(* Logix 5000 project; controller Carpenter_Meter_SCP vendor 1 type 14 code 217 rev 31.11; software revision 31.01; part 2 of 7 *)

ADD_ON_INSTRUCTION TGE_AI   (* revision 0.0, vendor Tallgrass Energy *)
VAR_IN_OUT
   UDT : TGE_AI_UDT; {required}
END_VAR
VAR_INPUT
   Raw : REAL; {required}   // Raw Data
END_VAR
VAR_OUTPUT
   EU : REAL; {access Read Only, visible}   // Scaled Value in Engineering Units
   Avg : REAL; {access Read Only, visible}   // Average value
   MalfAlm : BOOL; {access Read Only, visible}   // Signal Malfunction Alarm Status
   HAlm : BOOL; {access Read Only, visible}   // High Alarm status
   HHAlm : BOOL; {access Read Only, visible}   // High High Alarm status
   LAlm : BOOL; {access Read Only, visible}   // Low Alarm status
   LLAlm : BOOL; {access Read Only, visible}   // Low low Alarm status
   ROCNegAlm : BOOL; {access Read Only, visible}   // Negative Rate Of Change Alarm status
   ROCPosAlm : BOOL; {access Read Only, visible}   // Positive Rate Of Change Alarm status
   Percent : REAL; {access Read Only, visible}   // Percent of Engineering
END_VAR
VAR
   HHActive : BOOL;   // High High Alarm Active
   HActive : BOOL;   // High Alarm Active
   LActive : BOOL;   // Low Alarm Active
   LLActive : BOOL;   // Low Low Alarm Active
   RocAlm : TGE_ROC;
   MaxPriority : DINT; {access None}
END_VAR

ROUTINE Logic   (* ladder *)
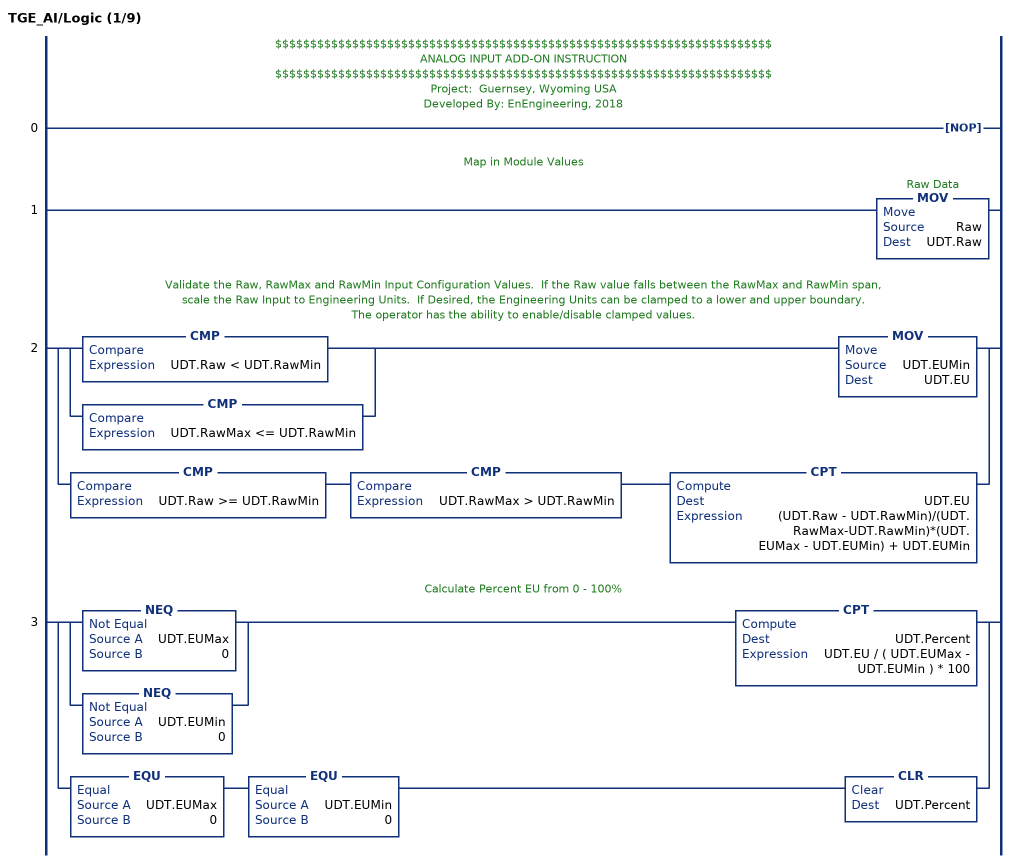
   // $$$$$$$$$$$$$$$$$$$$$$$$$$$$$$$$$$$$$$$$$$$$$$$$$$$$$$$$$$$$$$$$$$$$$$$
   // ANALOG INPUT ADD-ON INSTRUCTION
   // $$$$$$$$$$$$$$$$$$$$$$$$$$$$$$$$$$$$$$$$$$$$$$$$$$$$$$$$$$$$$$$$$$$$$$$
   // Project:  Guernsey, Wyoming USA
   // Developed By: EnEngineering, 2018
   0: NOP();
   // Map in Module Values
   1: MOV(Raw,UDT.Raw);
   // Validate the Raw, RawMax and RawMin Input Configuration Values.  If the Raw value falls between the RawMax and RawMin span,
   // scale the Raw Input to Engineering Units.  If Desired, the Engineering Units can be clamped to a lower and upper boundary.
   // The operator has the ability to enable/disable clamped values.
   2: [[CMP(UDT.Raw < UDT.RawMin) ,CMP(UDT.RawMax <= UDT.RawMin) ] MOV(UDT.EUMin,UDT.EU) ,CMP(UDT.Raw >= UDT.RawMin) CMP(UDT.RawMax > UDT.RawMin) CPT(UDT.EU,(UDT.Raw - UDT.RawMin)/(UDT.RawMax-UDT.RawMin)*(UDT.EUMax - UDT.EUMin) + UDT.EUMin) ];
   // Calculate Percent EU from 0 - 100%
   3: [[NEQ(UDT.EUMax,0) ,NEQ(UDT.EUMin,0) ] CPT(UDT.Percent,UDT.EU / ( UDT.EUMax - UDT.EUMin ) * 100) ,EQU(UDT.EUMax,0) EQU(UDT.EUMin,0) CLR(UDT.Percent) ];
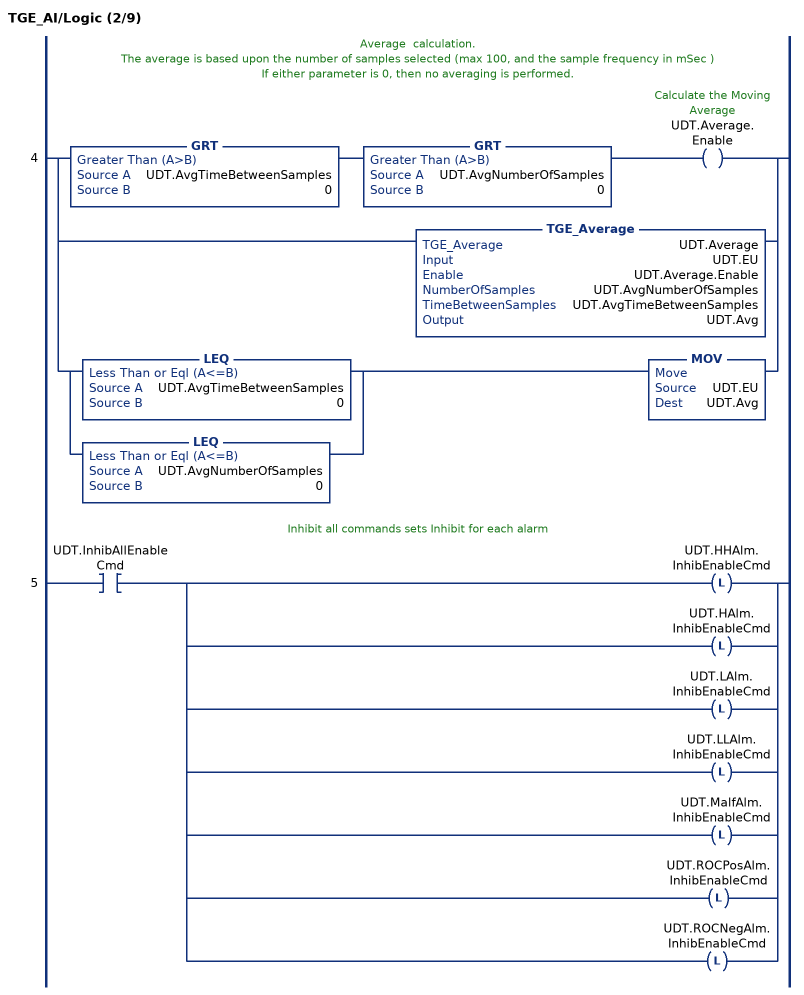
   // Average  calculation.
   // The average is based upon the number of samples selected (max 100, and the sample frequency in mSec )
   // If either parameter is 0, then no averaging is performed.
   4: [GRT(UDT.AvgTimeBetweenSamples,0) GRT(UDT.AvgNumberOfSamples,0) OTE(UDT.Average.Enable) ,TGE_Average(UDT.Average,UDT.EU,UDT.Average.Enable,UDT.AvgNumberOfSamples,UDT.AvgTimeBetweenSamples,UDT.Avg) ,[LEQ(UDT.AvgTimeBetweenSamples,0) ,LEQ(UDT.AvgNumberOfSamples,0) ] MOV(UDT.EU,UDT.Avg) ];
   // Inhibit all commands sets Inhibit for each alarm
   5: XIC(UDT.InhibAllEnableCmd)[OTL(UDT.HHAlm.InhibEnableCmd) ,OTL(UDT.HAlm.InhibEnableCmd) ,OTL(UDT.LAlm.InhibEnableCmd) ,OTL(UDT.LLAlm.InhibEnableCmd) ,OTL(UDT.MalfAlm.InhibEnableCmd) ,OTL(UDT.ROCPosAlm.InhibEnableCmd) ,OTL(UDT.ROCNegAlm.InhibEnableCmd) ];
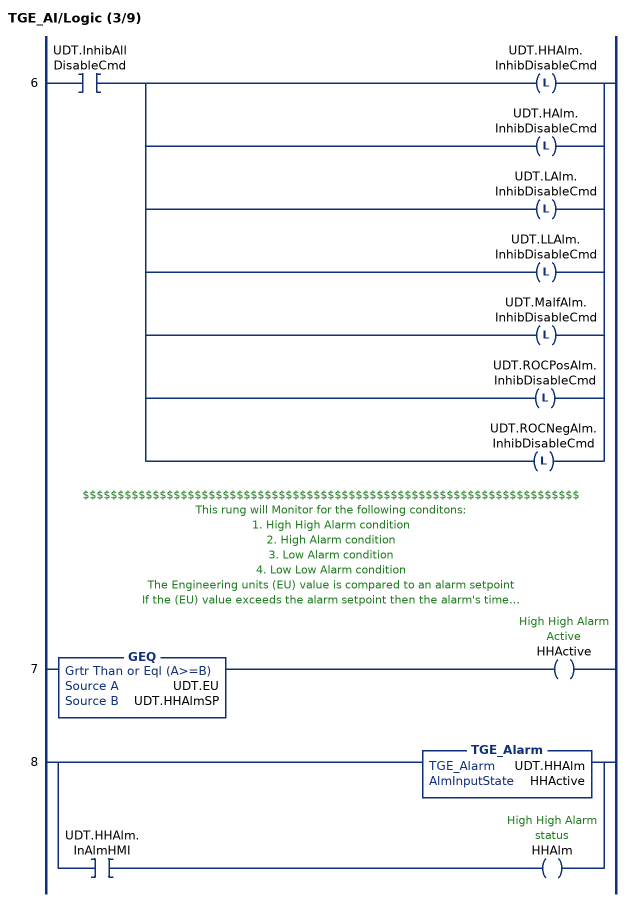
   6: XIC(UDT.InhibAllDisableCmd)[OTL(UDT.HHAlm.InhibDisableCmd) ,OTL(UDT.HAlm.InhibDisableCmd) ,OTL(UDT.LAlm.InhibDisableCmd) ,OTL(UDT.LLAlm.InhibDisableCmd) ,OTL(UDT.MalfAlm.InhibDisableCmd) ,OTL(UDT.ROCPosAlm.InhibDisableCmd) ,OTL(UDT.ROCNegAlm.InhibDisableCmd) ];
   // $$$$$$$$$$$$$$$$$$$$$$$$$$$$$$$$$$$$$$$$$$$$$$$$$$$$$$$$$$$$$$$$$$$$$$$
   //  This rung will Monitor for the following conditons:
   // 1. High High Alarm condition
   // 2. High Alarm condition
   // 3. Low Alarm condition
   // 4. Low Low Alarm condition
   // The Engineering units (EU) value is compared to an alarm setpoint
   //  If the (EU) value exceeds the alarm setpoint then the alarm's timer
   // preset value is loaded and the Alarm's Active bit is set
   // Note: The Preset value of this timer is configured via the udt
   // The alarm's Active bit is used as the Input to the aoiAlarm instruction.
   // The aoiAlarm's Alm bit is then used to update the Alarm status bit
   // $$$$$$$$$$$$$$$$$$$$$$$$$$$$$$$$$$$$$$$$$$$$$$$$$$$$$$$$$$$$$$$$$$$$$$$
   7: GEQ(UDT.EU,UDT.HHAlmSP)OTE(HHActive);
   8: [TGE_Alarm(UDT.HHAlm,HHActive) ,XIC(UDT.HHAlm.InAlmHMI) OTE(HHAlm) ];
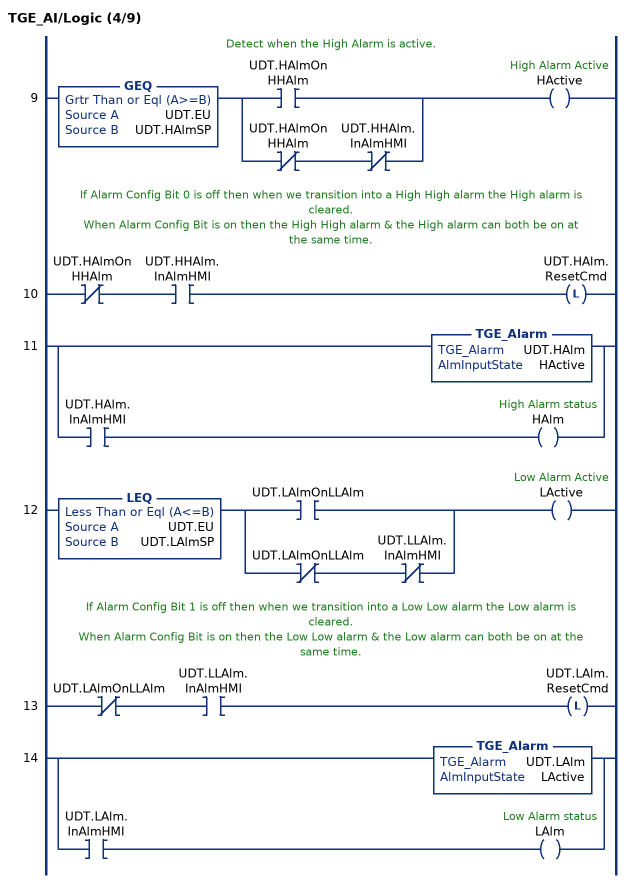
   // Detect when the High Alarm is active.
   9: GEQ(UDT.EU,UDT.HAlmSP)[XIC(UDT.HAlmOnHHAlm) ,XIO(UDT.HAlmOnHHAlm) XIO(UDT.HHAlm.InAlmHMI) ]OTE(HActive);
   // If Alarm Config Bit 0 is off then when we transition into a High High alarm the High alarm is cleared.
   // When Alarm Config Bit is on then the High High alarm & the High alarm can both be on at the same time.
   10: XIO(UDT.HAlmOnHHAlm)XIC(UDT.HHAlm.InAlmHMI)OTL(UDT.HAlm.ResetCmd);
   11: [TGE_Alarm(UDT.HAlm,HActive) ,XIC(UDT.HAlm.InAlmHMI) OTE(HAlm) ];
   12: LEQ(UDT.EU,UDT.LAlmSP)[XIC(UDT.LAlmOnLLAlm) ,XIO(UDT.LAlmOnLLAlm) XIO(UDT.LLAlm.InAlmHMI) ]OTE(LActive);
   // If Alarm Config Bit 1 is off then when we transition into a Low Low alarm the Low alarm is cleared.
   // When Alarm Config Bit is on then the Low Low alarm & the Low alarm can both be on at the same time.
   13: XIO(UDT.LAlmOnLLAlm)XIC(UDT.LLAlm.InAlmHMI)OTL(UDT.LAlm.ResetCmd);
   14: [TGE_Alarm(UDT.LAlm,LActive) ,XIC(UDT.LAlm.InAlmHMI) OTE(LAlm) ];
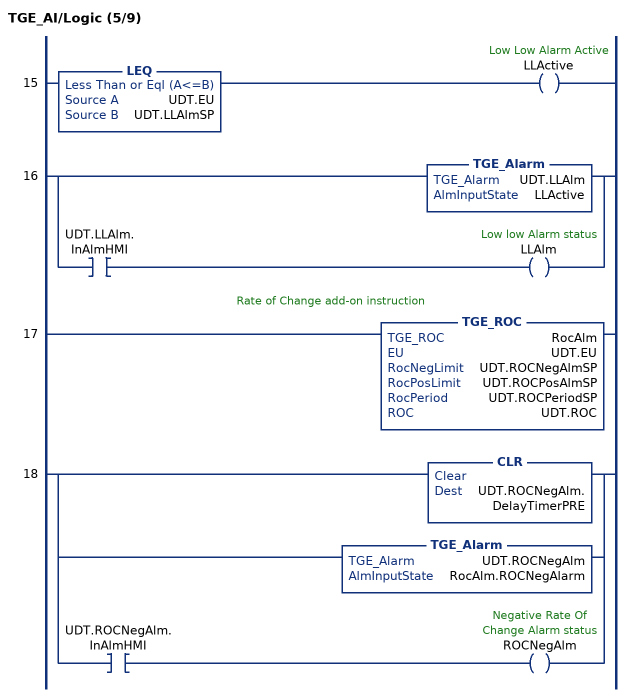
   15: LEQ(UDT.EU,UDT.LLAlmSP)OTE(LLActive);
   16: [TGE_Alarm(UDT.LLAlm,LLActive) ,XIC(UDT.LLAlm.InAlmHMI) OTE(LLAlm) ];
   // Rate of Change add-on instruction
   17: TGE_ROC(RocAlm,UDT.EU,UDT.ROCNegAlmSP,UDT.ROCPosAlmSP,UDT.ROCPeriodSP,UDT.ROC);
   18: [CLR(UDT.ROCNegAlm.DelayTimerPRE) ,TGE_Alarm(UDT.ROCNegAlm,RocAlm.ROCNegAlarm) ,XIC(UDT.ROCNegAlm.InAlmHMI) OTE(ROCNegAlm) ];
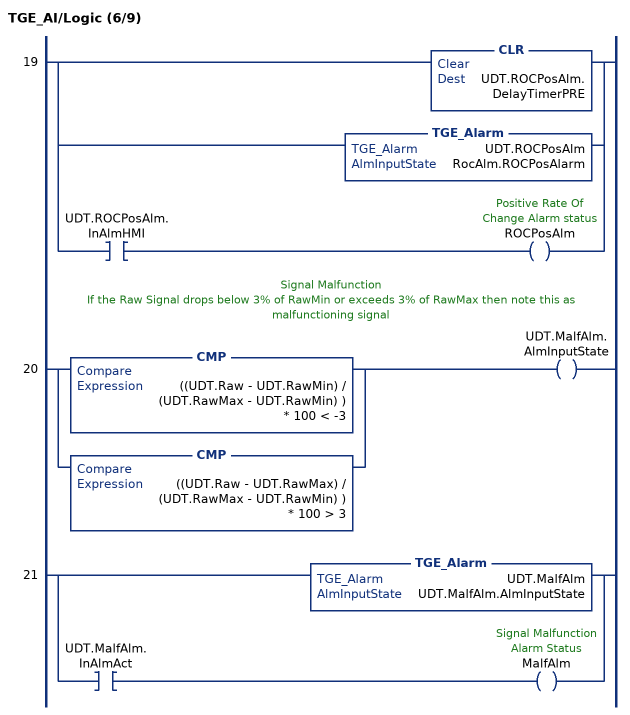
   19: [CLR(UDT.ROCPosAlm.DelayTimerPRE) ,TGE_Alarm(UDT.ROCPosAlm,RocAlm.ROCPosAlarm) ,XIC(UDT.ROCPosAlm.InAlmHMI) OTE(ROCPosAlm) ];
   // Signal Malfunction
   // If the Raw Signal drops below 3% of RawMin or exceeds 3% of RawMax then note this as malfunctioning signal
   20: [CMP(((UDT.Raw - UDT.RawMin) / (UDT.RawMax - UDT.RawMin) ) * 100 < -3) ,CMP(((UDT.Raw - UDT.RawMax) / (UDT.RawMax - UDT.RawMin) ) * 100 > 3) ]OTE(UDT.MalfAlm.AlmInputState);
   21: [TGE_Alarm(UDT.MalfAlm,UDT.MalfAlm.AlmInputState) ,XIC(UDT.MalfAlm.InAlmAct) OTE(MalfAlm) ];
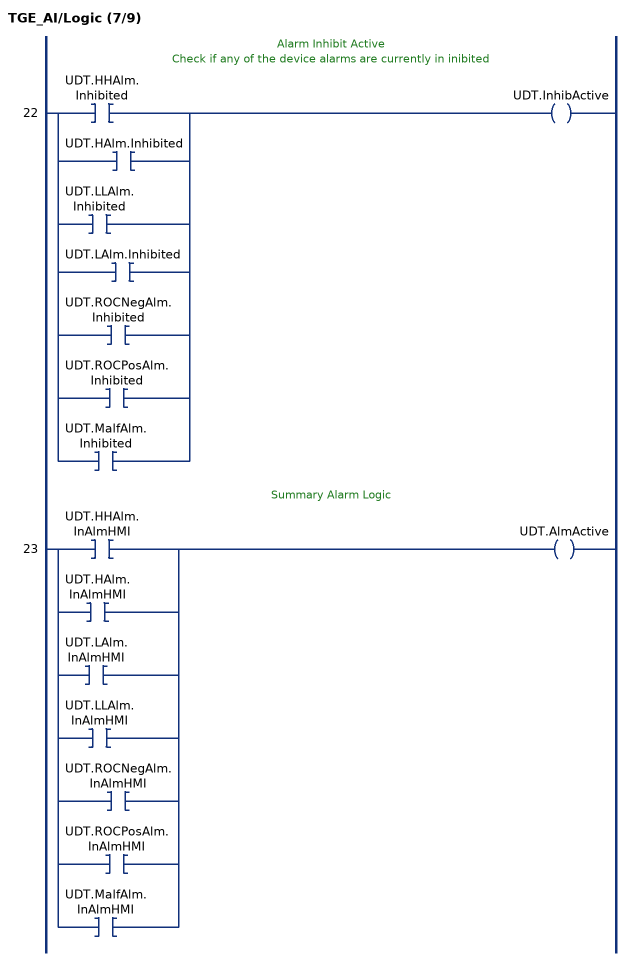
   // Alarm Inhibit Active
   // Check if any of the device alarms are currently in inibited
   22: [XIC(UDT.HHAlm.Inhibited) ,XIC(UDT.HAlm.Inhibited) ,XIC(UDT.LLAlm.Inhibited) ,XIC(UDT.LAlm.Inhibited) ,XIC(UDT.ROCNegAlm.Inhibited) ,XIC(UDT.ROCPosAlm.Inhibited) ,XIC(UDT.MalfAlm.Inhibited) ]OTE(UDT.InhibActive);
   // Summary Alarm Logic
   23: [XIC(UDT.HHAlm.InAlmHMI) ,XIC(UDT.HAlm.InAlmHMI) ,XIC(UDT.LAlm.InAlmHMI) ,XIC(UDT.LLAlm.InAlmHMI) ,XIC(UDT.ROCNegAlm.InAlmHMI) ,XIC(UDT.ROCPosAlm.InAlmHMI) ,XIC(UDT.MalfAlm.InAlmHMI) ]OTE(UDT.AlmActive);
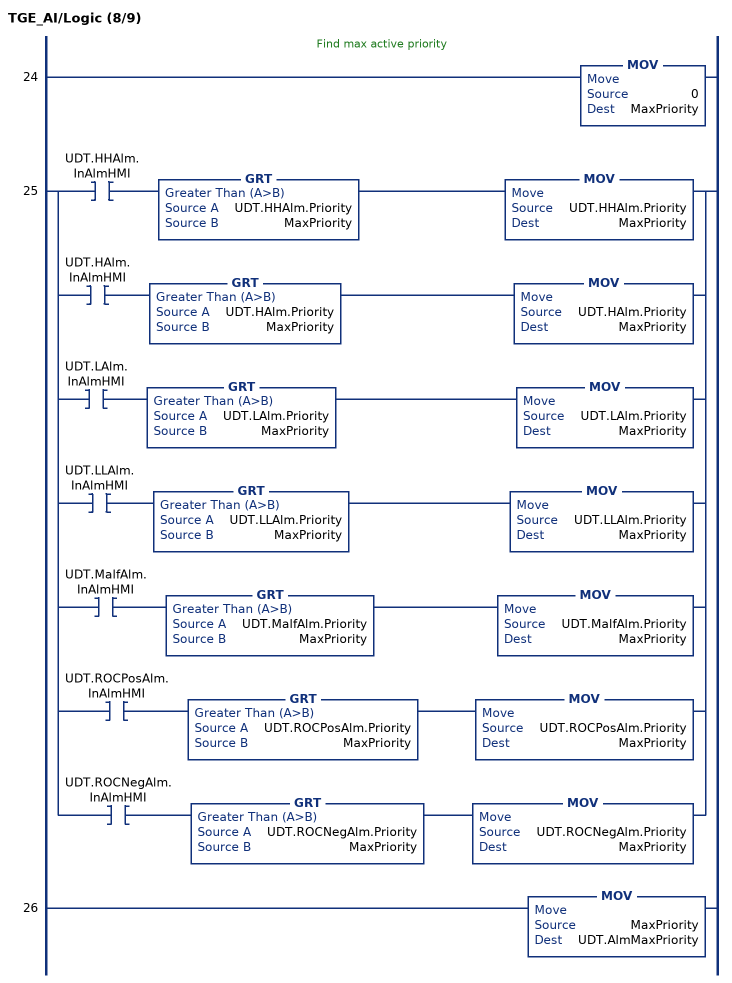
   // Find max active priority
   24: MOV(0,MaxPriority);
   25: [XIC(UDT.HHAlm.InAlmHMI) GRT(UDT.HHAlm.Priority,MaxPriority) MOV(UDT.HHAlm.Priority,MaxPriority) ,XIC(UDT.HAlm.InAlmHMI) GRT(UDT.HAlm.Priority,MaxPriority) MOV(UDT.HAlm.Priority,MaxPriority) ,XIC(UDT.LAlm.InAlmHMI) GRT(UDT.LAlm.Priority,MaxPriority) MOV(UDT.LAlm.Priority,MaxPriority) ,XIC(UDT.LLAlm.InAlmHMI) GRT(UDT.LLAlm.Priority,MaxPriority) MOV(UDT.LLAlm.Priority,MaxPriority) ,XIC(UDT.MalfAlm.InAlmHMI) GRT(UDT.MalfAlm.Priority,MaxPriority) MOV(UDT.MalfAlm.Priority,MaxPriority) ,XIC(UDT.ROCPosAlm.InAlmHMI) GRT(UDT.ROCPosAlm.Priority,MaxPriority) MOV(UDT.ROCPosAlm.Priority,MaxPriority) ,XIC(UDT.ROCNegAlm.InAlmHMI) GRT(UDT.ROCNegAlm.Priority,MaxPriority) MOV(UDT.ROCNegAlm.Priority,MaxPriority) ];
   26: MOV(MaxPriority,UDT.AlmMaxPriority);
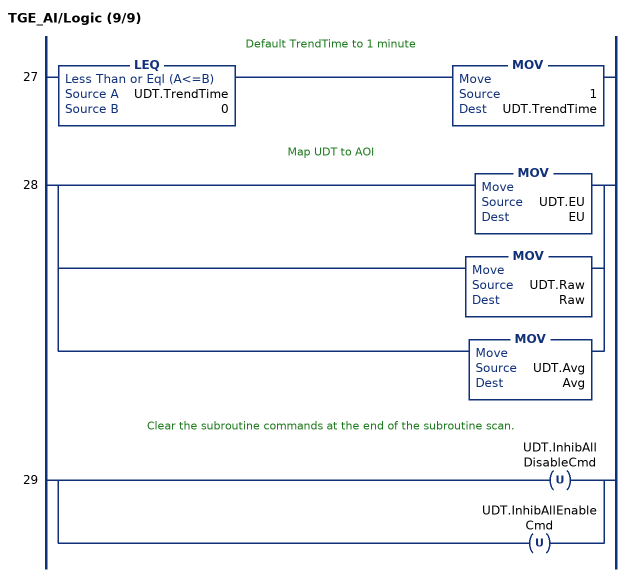
   // Default TrendTime to 1 minute
   27: LEQ(UDT.TrendTime,0)MOV(1,UDT.TrendTime);
   // Map UDT to AOI
   28: [MOV(UDT.EU,EU) ,MOV(UDT.Raw,Raw) ,MOV(UDT.Avg,Avg) ];
   // Clear the subroutine commands at the end of the subroutine scan.
   29: [OTU(UDT.InhibAllDisableCmd) ,OTU(UDT.InhibAllEnableCmd) ];
END_ROUTINE
END_ADD_ON_INSTRUCTION

ADD_ON_INSTRUCTION TGE_Alarm   (* revision 0.0, vendor Tallgrass Energy *)
VAR_INPUT
   EnableCmd : BOOL;
   DisableCmd : BOOL;
   ResetCmd : BOOL;
   TimerReset : BOOL;
   Enabled : BOOL; {visible}
   AckReq : BOOL;
   ResetReq : BOOL;
   AlmInputState : BOOL; {required}
   AckCmd : BOOL;
   AlmExists : BOOL := 1;
END_VAR
VAR_OUTPUT
   InAlmAct : BOOL; {visible}
END_VAR
VAR_INPUT
   InAlmHMI : BOOL;
END_VAR
VAR_OUTPUT
   Acked : BOOL;
END_VAR
VAR_INPUT
   DelayTimerPRE : REAL; {visible}
   ReminderTimerPRE : REAL; {visible}
END_VAR
VAR_OUTPUT
   ReminderFlag : BOOL; {visible}
   DelayTimerACC : REAL; {visible}
   ReminderTimerACC : REAL; {visible}
END_VAR
VAR_INPUT
   InhibEnableCmd : BOOL;
   InhibDisableCmd : BOOL;
END_VAR
VAR_OUTPUT
   Inhibited : BOOL;
   Priority : DINT; {visible}
END_VAR
VAR
   DelayTimer : TIMER;
   ReminderTimer : TIMER;
END_VAR

ROUTINE Logic   (* ladder *)
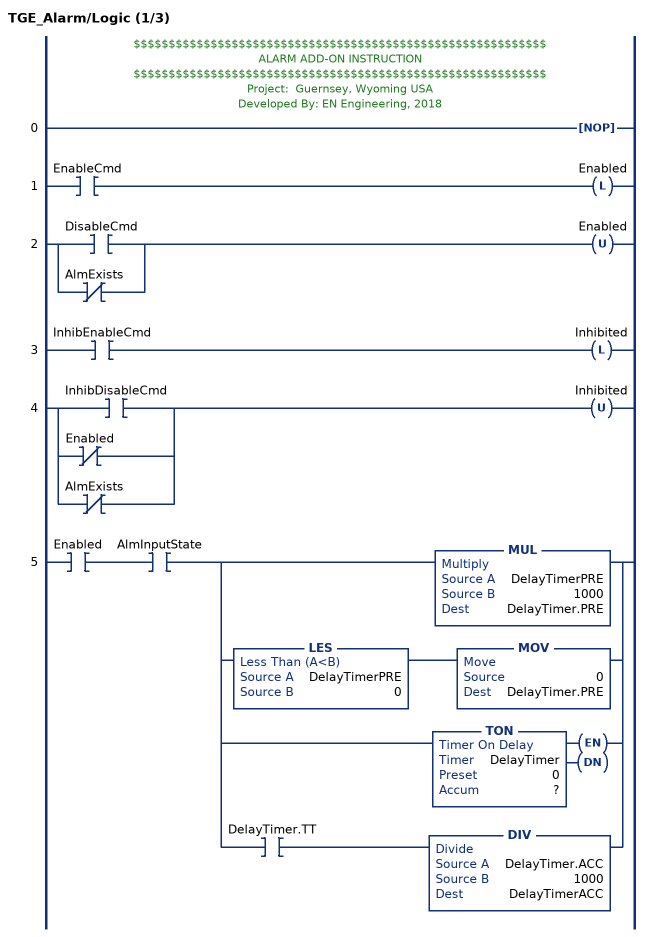
   // $$$$$$$$$$$$$$$$$$$$$$$$$$$$$$$$$$$$$$$$$$$$$$$$$$$$$$$$$$$
   // ALARM ADD-ON INSTRUCTION
   // $$$$$$$$$$$$$$$$$$$$$$$$$$$$$$$$$$$$$$$$$$$$$$$$$$$$$$$$$$$
   // Project:  Guernsey, Wyoming USA
   // Developed By: EN Engineering, 2018
   0: NOP();
   1: XIC(EnableCmd)OTL(Enabled);
   2: [XIC(DisableCmd) ,XIO(AlmExists) ]OTU(Enabled);
   3: XIC(InhibEnableCmd)OTL(Inhibited);
   4: [XIC(InhibDisableCmd) ,XIO(Enabled) ,XIO(AlmExists) ]OTU(Inhibited);
   5: XIC(Enabled)XIC(AlmInputState)[MUL(DelayTimerPRE,1000,DelayTimer.PRE) ,[LES(DelayTimerPRE,0) MOV(0,DelayTimer.PRE) ,TON(DelayTimer,?,?) ] ,XIC(DelayTimer.TT) DIV(DelayTimer.ACC,1000,DelayTimerACC) ];
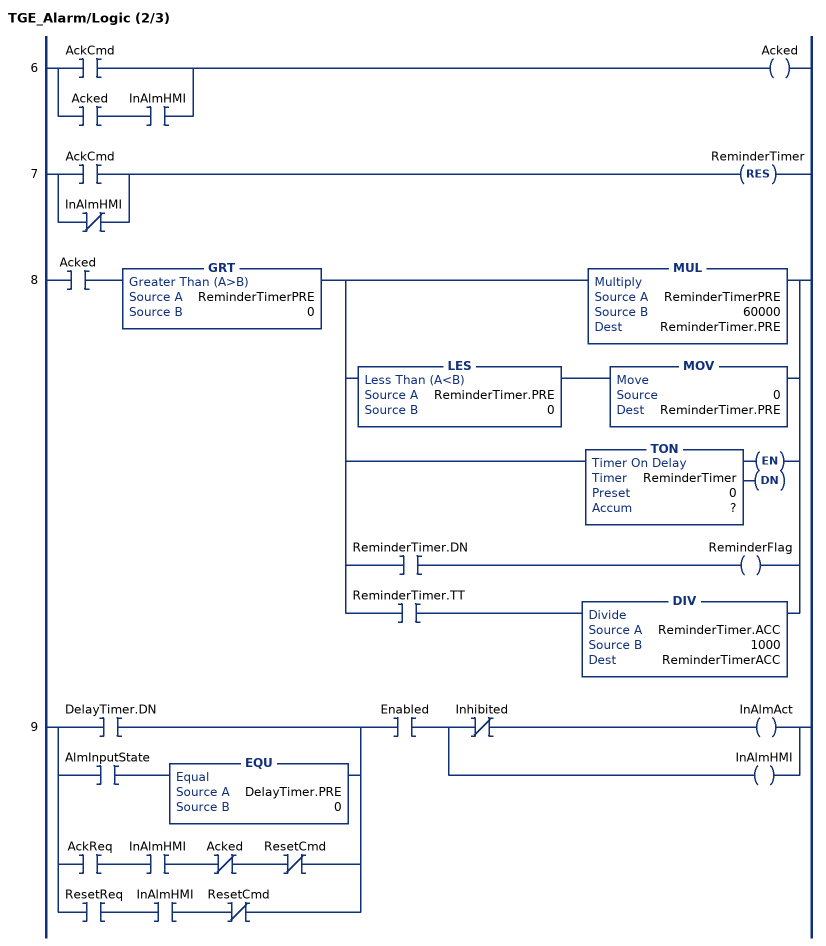
   6: [XIC(AckCmd) ,XIC(Acked) XIC(InAlmHMI) ]OTE(Acked);
   7: [XIC(AckCmd) ,XIO(InAlmHMI) ]RES(ReminderTimer);
   8: XIC(Acked)GRT(ReminderTimerPRE,0)[MUL(ReminderTimerPRE,60000,ReminderTimer.PRE) ,[LES(ReminderTimer.PRE,0) MOV(0,ReminderTimer.PRE) ,TON(ReminderTimer,?,?) ] ,XIC(ReminderTimer.DN) OTE(ReminderFlag) ,XIC(ReminderTimer.TT) DIV(ReminderTimer.ACC,1000,ReminderTimerACC) ];
   9: [[XIC(DelayTimer.DN) ,XIC(AlmInputState) EQU(DelayTimer.PRE,0) ] ,XIC(AckReq) XIC(InAlmHMI) XIO(Acked) XIO(ResetCmd) ,XIC(ResetReq) XIC(InAlmHMI) XIO(ResetCmd) ]XIC(Enabled)[XIO(Inhibited) OTE(InAlmAct) ,OTE(InAlmHMI) ];
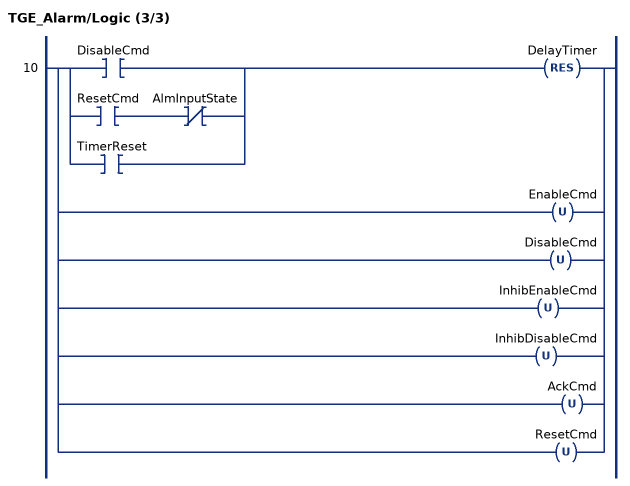
   10: [[XIC(DisableCmd) ,XIC(ResetCmd) XIO(AlmInputState) ,XIC(TimerReset) ] RES(DelayTimer) ,OTU(EnableCmd) ,OTU(DisableCmd) ,OTU(InhibEnableCmd) ,OTU(InhibDisableCmd) ,OTU(AckCmd) ,OTU(ResetCmd) ];
END_ROUTINE
END_ADD_ON_INSTRUCTION

ADD_ON_INSTRUCTION TGE_Average   (* revision 0.0, vendor Tallgrass Energy, ExecutePrescan *)
VAR_INPUT
   Input : REAL; {required}   // Analog Signal Input
   Enable : BOOL; {required}   // Calculate the Moving Average
   NumberOfSamples : DINT; {required}   // Number of Samples used in Calculation
   TimeBetweenSamples : DINT; {required}   // Time Between Samples in mSec
   SamplePulse : BOOL;   // Sample Pulse
END_VAR
VAR_OUTPUT
   Output : REAL; {access Read Only, required}   // Moving Average Output
END_VAR
VAR
   MAVE_01 : MOVING_AVERAGE := (SampleEnable := 1, NumberOfSamples := 1);
   TONR_01 : FBD_TIMER;
   OSRI_01 : FBD_ONESHOT;
   AverageArray : REAL[300];   // Average Array
   BNOT_01 : FBD_BOOLEAN_NOT := (In := 1);
   Real_Zero : REAL; {access None}
   ADD_01 : FBD_MATH; {access None}
   LES_01 : FBD_COMPARE; {access None}
   SEL_01 : SELECT; {access None}
   __l226943E508A92131 : BOOL; {access None}
   __l8BAE74C31515A0CC : REAL; {access None}
   __l8FE42AD99E759F48 : DINT; {access None}
   __l250EFCB3FE096DFA : BOOL; {access None}
   __l2717CE1F6A154822 : DINT; {access None}
END_VAR

ROUTINE Logic   (* function block diagram *)
   SHEET 1
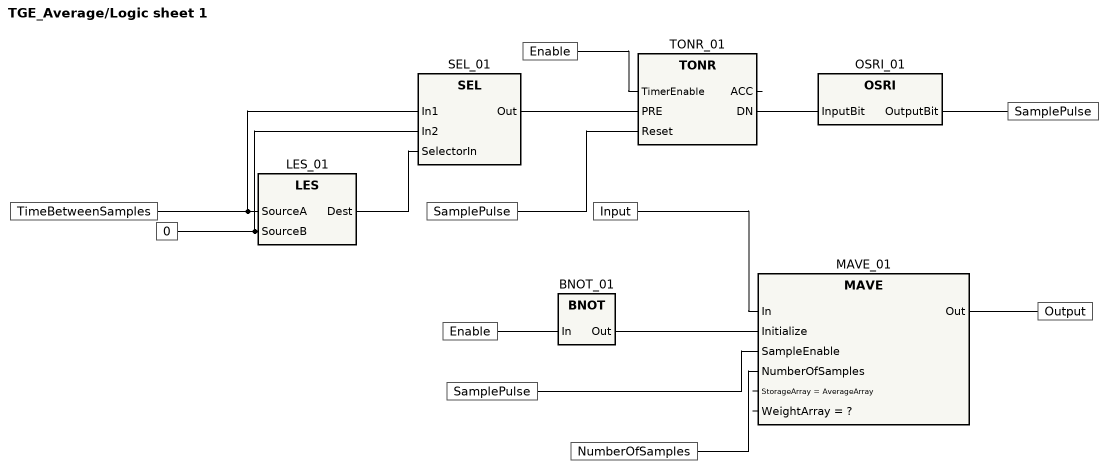
   LES_01 : LES(SourceA := TimeBetweenSamples, SourceB := 0);
   SEL_01 : SEL(In1 := TimeBetweenSamples, In2 := 0, SelectorIn := LES_01.Dest);
   BNOT_01 : BNOT(In := Enable);
   TONR_01 : TONR(TimerEnable := Enable, PRE := SEL_01.Out, Reset := SamplePulse);   // unwired pins: ACC
   MAVE_01 : MAVE(In := Input, Initialize := BNOT_01.Out, SampleEnable := SamplePulse, NumberOfSamples := NumberOfSamples, StorageArray := AverageArray, WeightArray := ?);
   OSRI_01 : OSRI(InputBit := TONR_01.DN);
   SamplePulse := OSRI_01.OutputBit;
   Output := MAVE_01.Out;
END_ROUTINE

ROUTINE Prescan   (* ladder *)
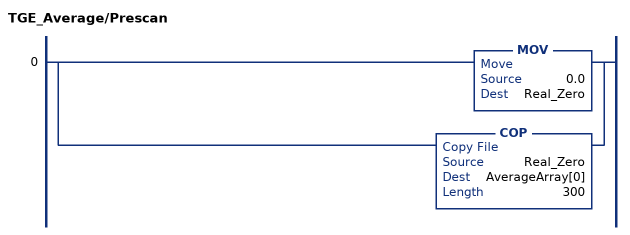
   0: [MOV(0.0,Real_Zero) ,COP(Real_Zero,AverageArray[0],300) ];
END_ROUTINE
END_ADD_ON_INSTRUCTION

ADD_ON_INSTRUCTION TGE_ROC   (* revision 0.0, vendor Tallgrass Energy *)
VAR_INPUT
   EU : REAL; {required}   // Engineering Units
   RocNegLimit : REAL; {required}   // Neg rate-of-change alarm limit in units per second
   RocPosLimit : REAL; {required}   // Pos rate-of-change alarm limit in units per second
   RocPeriod : REAL; {required}   // The time period used to evaluate the rate-of-change ala rms
END_VAR
VAR_OUTPUT
   ROC : REAL; {access Read Only, required}   // Rate of Change OutPut
   ROCPosAlarm : BOOL; {access Read Only, visible}   // Pos Rate of Change Alarm on
   ROCNegAlarm : BOOL; {access Read Only, visible}   // Neg Rate of Change Alarm on
END_VAR
VAR
   Alm : ALARM;
END_VAR

ROUTINE Logic   (* structured text *)
   /*
   $$$$$$$$$$$$$$$$$$$$$$$$$$$$$$$$$$$$$$$$$$$$$$$$$$$$$$$$$$$$$$
   			Rate of Change Add-on Instruction
   $$$$$$$$$$$$$$$$$$$$$$$$$$$$$$$$$$$$$$$$$$$$$$$$$$$$$$$$$$$$$$
   
    Project:  Hills Richmond Plant, Richmond, Indiana USA
   	   Developed By: Wheatland Systems, Inc. 2010			*/
   
   Alm.ROCPosLimit:=RocPosLimit;
   Alm.ROCNegLimit:=RocNegLimit;
   Alm.ROCPeriod:=RocPeriod;
   Alm.In:= EU;
   
   ALM(Alm);//Actually execute the Alarm instruction
   
   ROC:=Alm.ROC;
   ROCPosAlarm := Alm.ROCPosAlarm;
   ROCNegAlarm := Alm.ROCNegAlarm;
END_ROUTINE
END_ADD_ON_INSTRUCTION

ADD_ON_INSTRUCTION Valve_Control   (* revision 1.0, vendor Tallgrass Energy  *)
// Motor Operated Valve control logic
VAR_IN_OUT
   UDT : BaseVLVLiquid; {required}
END_VAR
VAR_INPUT
   Open_ILK : BOOL;   // Open Interlock
   Close_ILK : BOOL;   // Close Interlock
   sta_stat_vlv_start_req : BOOL;   // Station Start Valve Request
END_VAR
VAR_IN_OUT
   alarm_co : BOOL[32]; {required}
END_VAR
VAR_INPUT
   alarm_horn_req : BOOL; {required}
END_VAR
VAR_IN_OUT
   sta_stat : StaStatus; {required}
END_VAR
VAR_INPUT
   esd_active : BOOL;
   sys_plc_perm : BOOL;   // System PLC Permissive
END_VAR
VAR
   vlv_opn_req : BOOL; {access None}
END_VAR

ROUTINE Logic   (* ladder *)
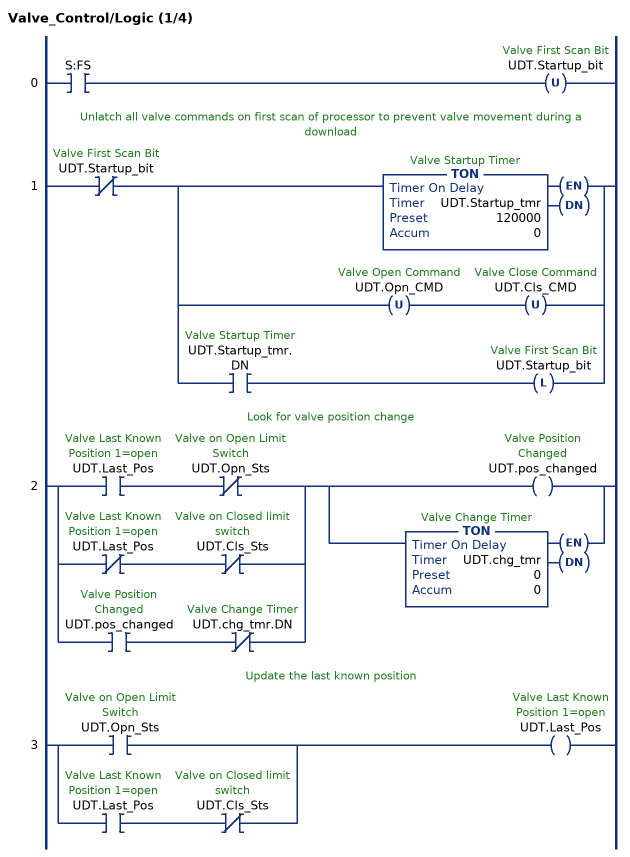
   0: XIC(S:FS)OTU(UDT.Startup_bit);
   // Unlatch all valve commands on first scan of processor to prevent valve movement during a download
   1: XIO(UDT.Startup_bit)[TON(UDT.Startup_tmr,120000,0) ,OTU(UDT.Opn_CMD) OTU(UDT.Cls_CMD) ,XIC(UDT.Startup_tmr.DN) OTL(UDT.Startup_bit) ];
   // Look for valve position change
   2: [XIC(UDT.Last_Pos) XIO(UDT.Opn_Sts) ,XIO(UDT.Last_Pos) XIO(UDT.Cls_Sts) ,XIC(UDT.pos_changed) XIO(UDT.chg_tmr.DN) ][OTE(UDT.pos_changed) ,TON(UDT.chg_tmr,0,0) ];
   // Update the last known position
   3: [XIC(UDT.Opn_Sts) ,XIC(UDT.Last_Pos) XIO(UDT.Cls_Sts) ]OTE(UDT.Last_Pos);
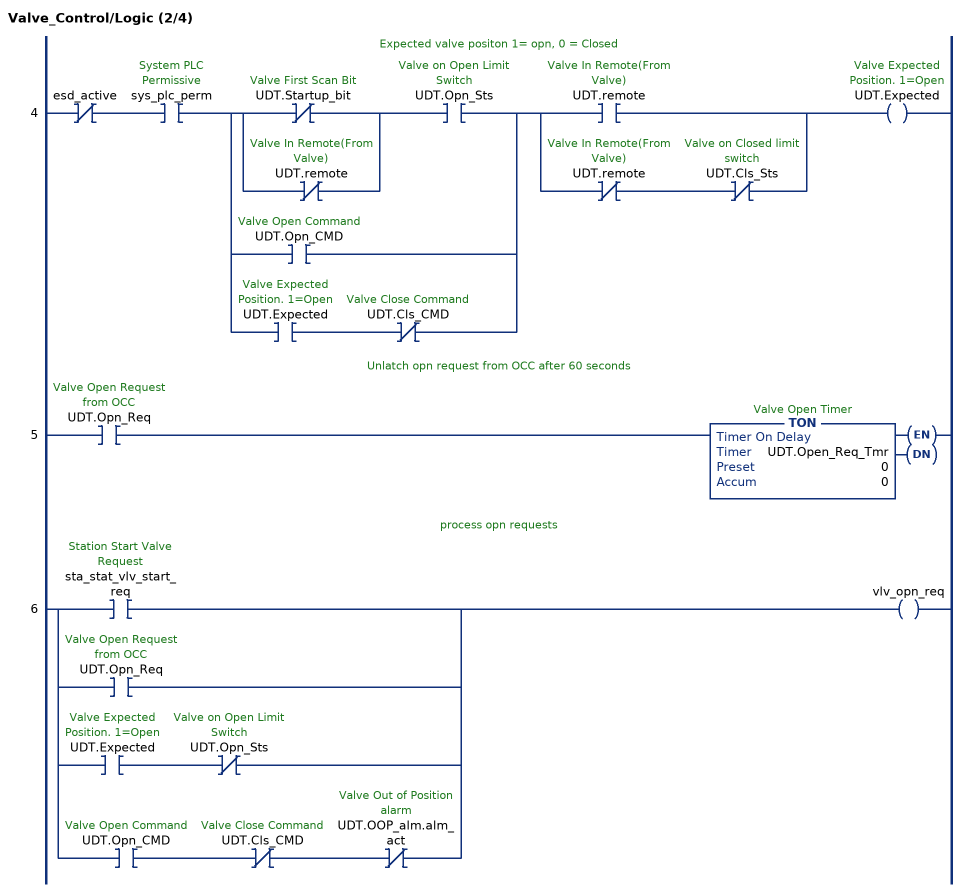
   // Expected valve positon 1= opn, 0 = Closed
   4: XIO(esd_active)XIC(sys_plc_perm)[[XIO(UDT.Startup_bit) ,XIO(UDT.remote) ] XIC(UDT.Opn_Sts) ,XIC(UDT.Opn_CMD) ,XIC(UDT.Expected) XIO(UDT.Cls_CMD) ][XIC(UDT.remote) ,XIO(UDT.remote) XIO(UDT.Cls_Sts) ]OTE(UDT.Expected);
   // Unlatch opn request from OCC after 60 seconds
   5: XIC(UDT.Opn_Req)TON(UDT.Open_Req_Tmr,0,0);
   // process opn requests
   6: [XIC(sta_stat_vlv_start_req) ,XIC(UDT.Opn_Req) ,XIC(UDT.Expected) XIO(UDT.Opn_Sts) ,XIC(UDT.Opn_CMD) XIO(UDT.Cls_CMD) XIO(UDT.OOP_alm.alm_act) ]OTE(vlv_opn_req);
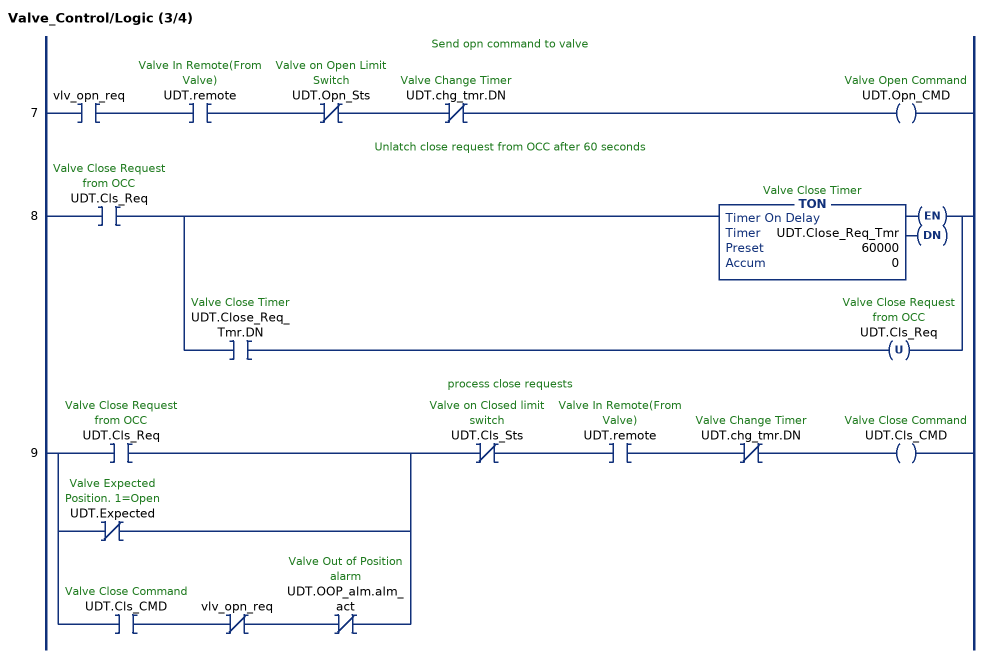
   // Send opn command to valve
   7: XIC(vlv_opn_req)XIC(UDT.remote)XIO(UDT.Opn_Sts)XIO(UDT.chg_tmr.DN)OTE(UDT.Opn_CMD);
   // Unlatch close request from OCC after 60 seconds
   8: XIC(UDT.Cls_Req)[TON(UDT.Close_Req_Tmr,60000,0) ,XIC(UDT.Close_Req_Tmr.DN) OTU(UDT.Cls_Req) ];
   // process close requests
   9: [XIC(UDT.Cls_Req) ,XIO(UDT.Expected) ,XIC(UDT.Cls_CMD) XIO(vlv_opn_req) XIO(UDT.OOP_alm.alm_act) ]XIO(UDT.Cls_Sts)XIC(UDT.remote)XIO(UDT.chg_tmr.DN)OTE(UDT.Cls_CMD);
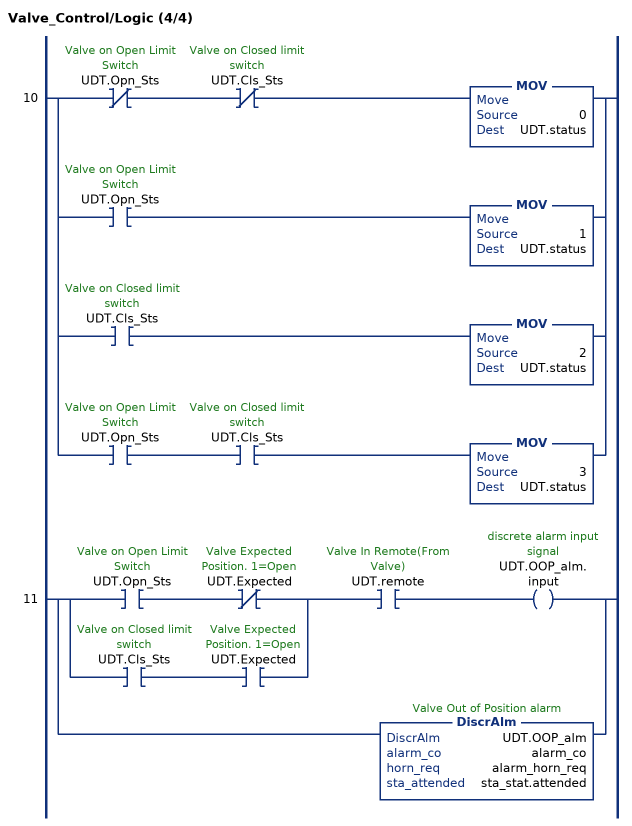
   10: [XIO(UDT.Opn_Sts) XIO(UDT.Cls_Sts) MOV(0,UDT.status) ,XIC(UDT.Opn_Sts) MOV(1,UDT.status) ,XIC(UDT.Cls_Sts) MOV(2,UDT.status) ,XIC(UDT.Opn_Sts) XIC(UDT.Cls_Sts) MOV(3,UDT.status) ];
   11: [[XIC(UDT.Opn_Sts) XIO(UDT.Expected) ,XIC(UDT.Cls_Sts) XIC(UDT.Expected) ] XIC(UDT.remote) OTE(UDT.OOP_alm.input) ,DiscrAlm(UDT.OOP_alm,alarm_co,alarm_horn_req,sta_stat.attended) ];
END_ROUTINE
END_ADD_ON_INSTRUCTION
